TYPE ST_NeutralTransformer_events :
STRUCT
	b_TemperatureHighPhase						: ARRAY [1..3] OF BOOL; //1=L1, 2=L2, 3=L3
	b_TemperatureTooHighPhase					: ARRAY [1..3] OF BOOL; //1=L1, 2=L2, 3=L3
	b_VoltageUnbalanceHigh										: BOOL;
	b_VoltageUnbalanceTooHigh									: BOOL;
	b_NeutralCurrentHigh										: BOOL;
	b_NeutralCurrentTooHigh										: BOOL;
	
END_STRUCT
END_TYPE

(* stored: Version 1.1.0.1, ProductVersion 3.1.4026.18
   DUT ST_NeutralTransformer_events: Id {5983dfa5-e638-4b61-9d5f-8062ac9d1d0b} *)
